// TIA Portal V19 export
DATA_BLOCK "BATCH DATA"   // DB171
{ S7_Optimized_Access := 'FALSE' }
   VAR
      PRODUCT_NAME : String[30] := '  PRODUCT NAME             :  ';
      PRODUCT_NAME_CONCATE : String[80];
      BATCH_NO : String[30] := '  BATCH NO                 :  ';
      BATCH_NO_CONCATE : String[80];
      EQUIPMENT_ID_NO : String[30] := '  EQUIPMENT ID NO          :  ';
      EQUIPMENT_ID_NO_CONCATE : String[80];
      RECIPE_NO : String[30] := '  RECIPE NO                :  ';
      RECIPE_NO_CONCATE : String[80];
      OPERATOR_NAME : String[30] := '  OPERATOR NAME            :  ';
      OPERATOR_NAME_CONCATE : String[80];
      EMPLOYE_CODE : String[30] := '  EMPLOYE CODE             :  ';
      EMPLOYE_CODE_CONCATE : String[80];
   END_VAR
BEGIN
END_DATA_BLOCK
